// Mitsubishi GX Works2 project: plc2   PLC: Q03UDV

PROGRAM MAIN
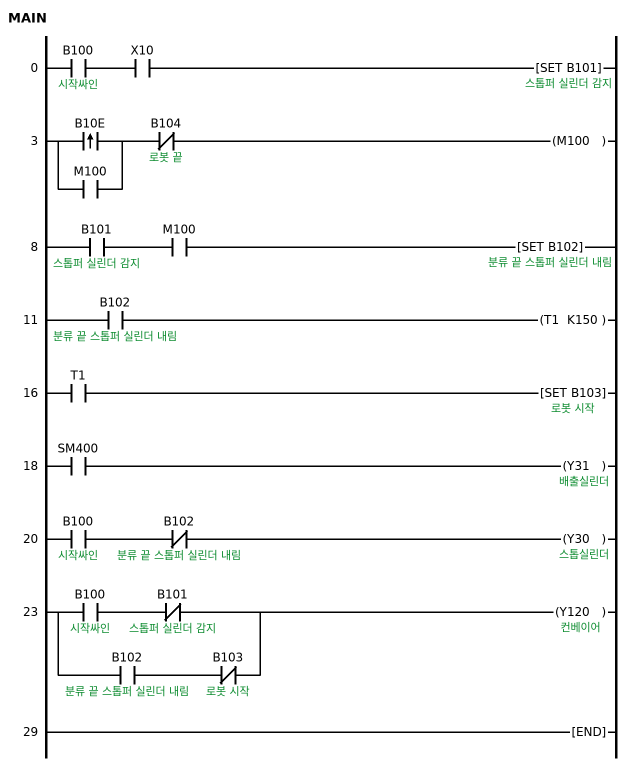
0     LD      B100  ; 시작싸인
      AND     X10
      SET     B101  ; 스톱퍼 실린더 감지
3     LDP     B10E
      OR      M100
      ANI     B104  ; 로봇 끝
      OUT     M100
8     LD      B101  ; 스톱퍼 실린더 감지
      AND     M100
      SET     B102  ; 분류 끝 스톱퍼 실린더 내림
11    LD      B102  ; 분류 끝 스톱퍼 실린더 내림
      OUT     T1 K150
16    LD      T1
      SET     B103  ; 로봇 시작
18    LD      SM400
      OUT     Y31  ; 배출실린더
20    LD      B100  ; 시작싸인
      ANI     B102  ; 분류 끝 스톱퍼 실린더 내림
      OUT     Y30  ; 스톱실린더
23    LD      B100  ; 시작싸인
      ANI     B101  ; 스톱퍼 실린더 감지
      LD      B102  ; 분류 끝 스톱퍼 실린더 내림
      ANI     B103  ; 로봇 시작
      ORB
      OUT     Y120  ; 컨베이어
29    END
END_PROGRAM
